FUNCTION_BLOCK FB_ValveCtrl32
VAR_INPUT
	i_Interlocks		:ARRAY[1..8] OF BOOL;
	i_ProcesslocksOK	:BOOL;
	i_AutoCmd			:BOOL;
	i_ManCmd			:BOOL;
	i_ServiceMode		:BOOL;
	i_EnableHP			:BOOL;
	i_EnableWP			:BOOL;
	i_HP				:BOOL;
	i_WP				:BOOL;
	i_Timeout			:INT;
	i_MaintLimit		:UDINT;
	i_PresetValue		:UDINT;
	i_WritePreset		:BOOL;
END_VAR
VAR_OUTPUT
	q_InterlocksOK		:BOOL;
	q_Enabled			:BOOL;
	q_Cmd				:BOOL;
	q_Traveling			:BOOL;
	q_AtHP				:BOOL;
	q_AtWP				:BOOL;
	q_TimeoutHP			:BOOL;
	q_TimeoutWP			:BOOL;
	q_SensorsFlt		:BOOL;
	q_TotalCycles		:UDINT;
	q_MaintCycles		:UDINT;
	q_MaintenanceCall	:BOOL;
	q_State				:INT;
END_VAR
VAR
	tonTimeoutHP		:TON;
	tonTimeoutWP		:TON;
	tonSensorsFlt		:TON;
	tofDelayOut			:TOF;
	bCmd				:BOOL;
END_VAR
VAR // added by the converter: edge detectors and wires of the graphical bodies
    _rt1, _rt2 : R_TRIG;
    _w1 : BOOL;
END_VAR

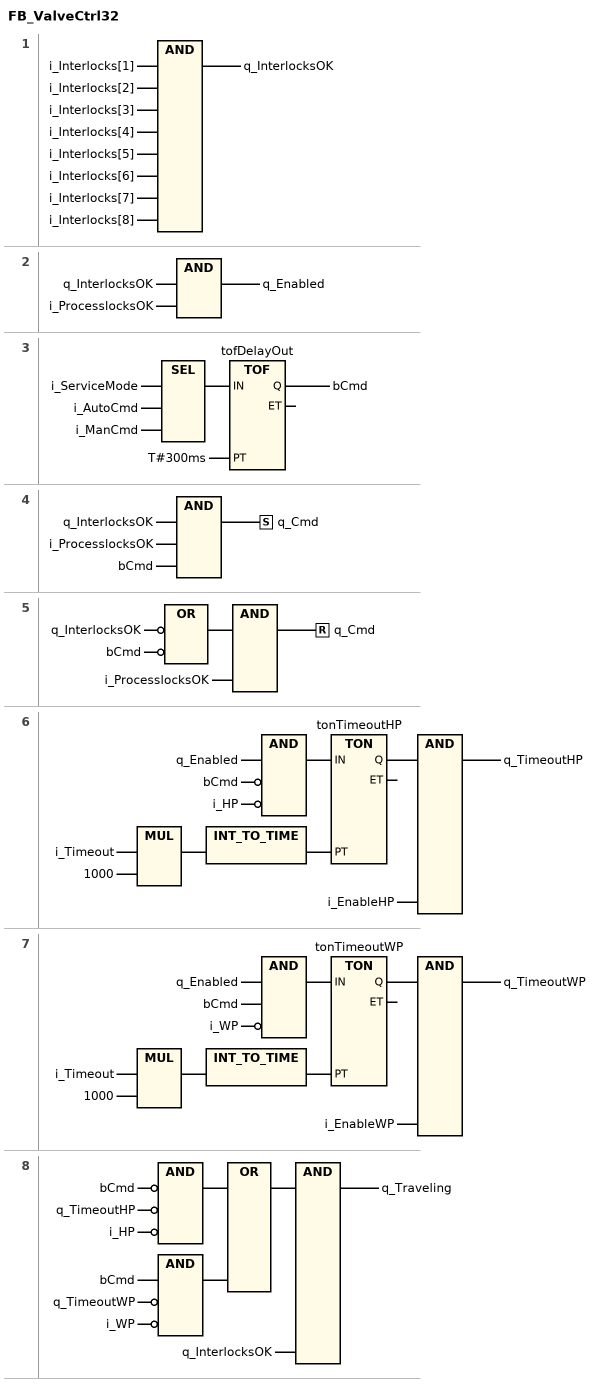
// NETWORK 1
q_InterlocksOK := i_Interlocks[1] AND i_Interlocks[2] AND i_Interlocks[3] AND i_Interlocks[4] AND i_Interlocks[5] AND i_Interlocks[6] AND i_Interlocks[7] AND i_Interlocks[8];

// NETWORK 2
q_Enabled := q_InterlocksOK AND i_ProcesslocksOK;

// NETWORK 3
tofDelayOut(IN := SEL(i_ServiceMode, i_AutoCmd, i_ManCmd), PT := T#300ms); // TOF
bCmd := tofDelayOut.Q;

// NETWORK 4
q_Cmd S= q_InterlocksOK AND i_ProcesslocksOK AND bCmd;

// NETWORK 5
q_Cmd R= (NOT q_InterlocksOK OR NOT bCmd) AND i_ProcesslocksOK;

// NETWORK 6
tonTimeoutHP(IN := q_Enabled AND NOT bCmd AND NOT i_HP, PT := INT_TO_TIME(i_Timeout * 1000)); // TON
q_TimeoutHP := tonTimeoutHP.Q AND i_EnableHP;

// NETWORK 7
tonTimeoutWP(IN := q_Enabled AND bCmd AND NOT i_WP, PT := INT_TO_TIME(i_Timeout * 1000)); // TON
q_TimeoutWP := tonTimeoutWP.Q AND i_EnableWP;

// NETWORK 8
q_Traveling := (NOT bCmd AND NOT q_TimeoutHP AND NOT i_HP OR bCmd AND NOT q_TimeoutWP AND NOT i_WP) AND q_InterlocksOK;

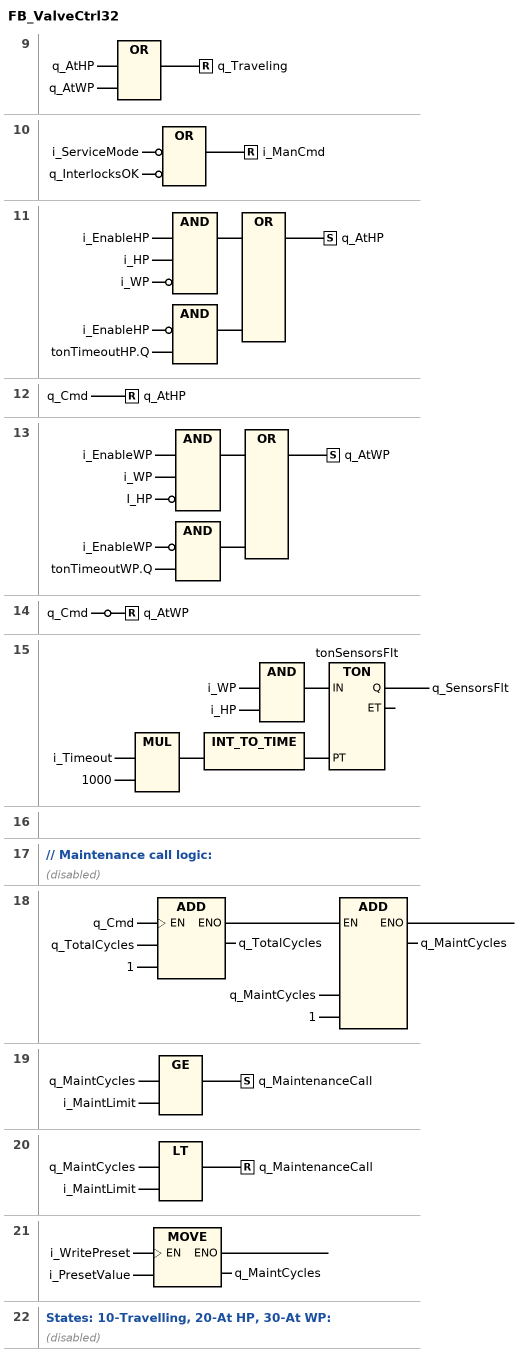
// NETWORK 9
q_Traveling R= q_AtHP OR q_AtWP;

// NETWORK 10
i_ManCmd R= NOT i_ServiceMode OR NOT q_InterlocksOK;

// NETWORK 11
q_AtHP S= i_EnableHP AND i_HP AND NOT i_WP OR NOT i_EnableHP AND tonTimeoutHP.Q;

// NETWORK 12
q_AtHP R= q_Cmd;

// NETWORK 13
q_AtWP S= i_EnableWP AND i_WP AND NOT I_HP OR NOT i_EnableWP AND tonTimeoutWP.Q;

// NETWORK 14
q_AtWP R= NOT q_Cmd;

// NETWORK 15
tonSensorsFlt(IN := i_WP AND i_HP, PT := INT_TO_TIME(i_Timeout * 1000)); // TON
q_SensorsFlt := tonSensorsFlt.Q;

// NETWORK 16

// NETWORK 17 (disabled)
// label: // Maintenance call logic

// NETWORK 18
_rt1(CLK := q_Cmd);
_w1 := _rt1.Q;
IF _w1 THEN q_TotalCycles := q_TotalCycles + 1; END_IF
IF _w1 THEN q_MaintCycles := q_MaintCycles + 1; END_IF

// NETWORK 19
q_MaintenanceCall S= q_MaintCycles >= i_MaintLimit;

// NETWORK 20
q_MaintenanceCall R= q_MaintCycles < i_MaintLimit;

// NETWORK 21
_rt2(CLK := i_WritePreset);
IF _rt2.Q THEN q_MaintCycles := i_PresetValue; END_IF

// NETWORK 22 (disabled)
// label: States: 10-Travelling, 20-At HP, 30-At WP

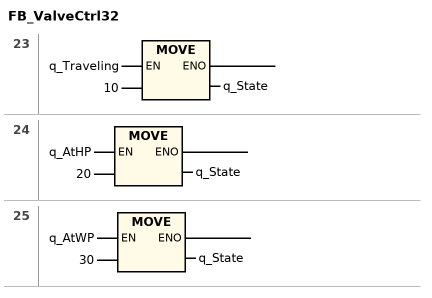
// NETWORK 23
IF q_Traveling THEN q_State := 10; END_IF

// NETWORK 24
IF q_AtHP THEN q_State := 20; END_IF

// NETWORK 25
IF q_AtWP THEN q_State := 30; END_IF

END_FUNCTION_BLOCK

(* stored: Version 1.1.0.1, ProductVersion 3.1.4024.12
   POU FB_ValveCtrl32: Id {fc1aceea-8c12-42d0-b807-9e9f2f1827d9}, SpecialFunc None *)
